// TIA Portal V17 export
// export: Created 2022-03-12T16:05:28.998489Z, ExportSetting WithDefaults, DisplayName Totally Integrated Automation Portal, DisplayVersion V17, DisplayName TIA Portal Openness, DisplayVersion V17, DisplayName TIA Portal Version Control Interface, DisplayVersion V17, DisplayName STEP 7 Professional, DisplayVersion V17, DisplayName STEP 7 Safety, DisplayVersion V17, DisplayName WinCC Advanced / Unified PC, DisplayVersion V17
DATA_BLOCK "EM01"   // DB31669
TITLE = EM01
{ S7_Optimized_Access := 'TRUE' }
AUTHOR : tech.team.motioncontrol@siemens.com
FAMILY : CPG
VERSION : 1.0
// Support: tech.team.motioncontrol@siemens.com
// Fax: +49 (0) 9131/98-1297
// stored: AutoNumber true, DBAccessibleFromOPCUA true, DBAccessibleFromWebserver true, IsOnlyStoredInLoadMemory false, IsRetainMemResEnabled false, IsWriteProtectedInAS false, MemoryReserve 100
   VAR
      PackML_Sts { ExternalWritable := 'False'} : Struct   // PackML Module Status - EM and all control modules
         Unit { ExternalWritable := 'False'; S7_SetPoint := 'True'} : "CPG_typePackML_ModuleSts";   // PackML Module Status - EM - master status
         Alarm { ExternalWritable := 'False'; S7_SetPoint := 'True'} : "CPG_typePackML_ModuleSts";   // PackML Module Status - alarm status
         CM01 { ExternalWritable := 'False'; S7_SetPoint := 'True'} : "CPG_typePackML_ModuleSts";   // PackML Module Status - CM 01
         CM02 { ExternalWritable := 'False'; S7_SetPoint := 'True'} : "CPG_typePackML_ModuleSts";   // PackML Module Status - CM 02
         CM03 { ExternalWritable := 'False'; S7_SetPoint := 'True'} : "CPG_typePackML_ModuleSts";   // PackML Module Status - CM 03
         CM04 { ExternalWritable := 'False'; S7_SetPoint := 'True'} : "CPG_typePackML_ModuleSts";   // PackML Module Status - CM 04
         CM05 { ExternalWritable := 'False'; S7_SetPoint := 'True'} : "CPG_typePackML_ModuleSts";   // PackML Module Status - CM 05
         CM06 { ExternalWritable := 'False'; S7_SetPoint := 'True'} : "CPG_typePackML_ModuleSts";   // PackML Module Status - CM 06
         CM07 { ExternalWritable := 'False'; S7_SetPoint := 'True'} : "CPG_typePackML_ModuleSts";   // PackML Module Status - CM 07
         CM08 { ExternalWritable := 'False'; S7_SetPoint := 'True'} : "CPG_typePackML_ModuleSts";   // PackML Module Status - CM 08
         CM09 { ExternalWritable := 'False'; S7_SetPoint := 'True'} : "CPG_typePackML_ModuleSts";   // PackML Module Status - CM 09
         CM10 { ExternalWritable := 'False'; S7_SetPoint := 'True'} : "CPG_typePackML_ModuleSts";   // PackML Module Status - CM 10
      END_STRUCT;
      Alarm { ExternalAccessible := 'False'; ExternalVisible := 'False'; ExternalWritable := 'False'; S7_SetPoint := 'True'} : "CPG_typeEventStatus";   // Alarm Event Status - EM01 Status
      Warning { ExternalAccessible := 'False'; ExternalVisible := 'False'; ExternalWritable := 'False'; S7_SetPoint := 'True'} : "CPG_typeEventStatus";   // Warning Event Status - EM01 Status
      Status { ExternalAccessible := 'False'; ExternalVisible := 'False'; ExternalWritable := 'False'; S7_SetPoint := 'True'} : "CPG_typeEventStatus";   // Event Status - EM01 Status
   END_VAR
BEGIN
END_DATA_BLOCK
